{attribute addProperty BoxType "AT2050-0501-0020"}
{attribute addProperty Id "A_0087_AT2050_5501_0016_AT2050_5501AT2050_3DCFC8D064080"}
{attribute addProperty CRC "1961037632"}
{attribute addProperty SizeInBites "640"}
{attribute addProperty SizeInBytes "80"}
TYPE A_0057_AT2050_0501_0020_74E30F40 EXTENDS AT2050_9506A482 :
STRUCT
	{attribute addProperty Name "A_0087_AT2050_5501_0016_AT2050_5501"}
	A_0087_AT2050_5501_0016_AT2050_5501 : AT2050_3DCFC8D0;
END_STRUCT
END_TYPE

(* stored: Version 1.2.0.0, ProductVersion 3.1.4024.9
   DUT A_0057_AT2050_0501_0020_74E30F40: Id {6e153d13-a860-4beb-9e9e-49e27c2c7546} *)
